(* Logix 5000 project; controller Savage_Saw vendor 1 type 14 code 152 rev 33.11; software revision 33.04 *)

TASK MainTask (continuous, watchdog 500 ms) : MainProgram

MODULES
   Local : vendor 1 type 14 code 152 (PointIO 0, rev 33.11)
      Kane : vendor 590 type 43 code 5 (Ethernet 192.168.1.11, rev 1.1, StandardDataDriven RPI 20 ms)
      Discrete_IO : Embedded (PointIO 1, rev 33.11, Output RPI 20 ms)
END_MODULES

TYPE Kane_OUT_DATA1 :
STRUCT
   Unassigned_Var_Table_12 : REAL;
   Unassigned_Var_Table_13 : REAL;
   Unassigned_Var_Table_14 : REAL;
   Unassigned_Var_Table_15 : REAL;
   Unassigned_Var_Table_16 : REAL;
   Unassigned_Var_Table_17 : REAL;
   Unassigned_Var_Table_18 : REAL;
   Unassigned_Var_Table_19 : REAL;
   Unassigned_Var_Table_20 : REAL;
   Unassigned_Var_Table_21 : REAL;
END_STRUCT
END_TYPE

TYPE RMC_IN :
STRUCT
   xCutStatus : DINT;
   yBedStatus : DINT;
   zDepthStatus : DINT;
   xCutPosition : REAL;
   yBedPosition : REAL;
   zDepthPosition : REAL;
END_STRUCT
END_TYPE

TYPE RMC_OUT :
STRUCT
   xCutPosnCommand : REAL;
   yBedPosnCommand : REAL;
   zDepthPosnCommand : REAL;
   xCutVelocity : REAL;
   yBedVelocity : REAL;
   zDepthVelocity : REAL;
END_STRUCT
END_TYPE

VAR_GLOBAL   (* controller tags *)
   RMC_Busy : BOOL;
   RMC_In : RMC_IN := (xCutStatus := 67154500, yBedStatus := 67117633, zDepthStatus := 67121732, xCutPosition := 15.000001, yBedPosition := 10.0, zDepthPosition := 18.928001);
   RMC_Out : RMC_OUT := (xCutPosnCommand := 9.999, yBedPosnCommand := 2.2, zDepthPosnCommand := 3.3, xCutVelocity := 4.4, yBedVelocity := 5.5, zDepthVelocity := 69.6);
   RMC_SendRequest : BOOL;
END_VAR

PROGRAM MainProgram   (* main routine RMC *)

ROUTINE RMC   (* ladder *)
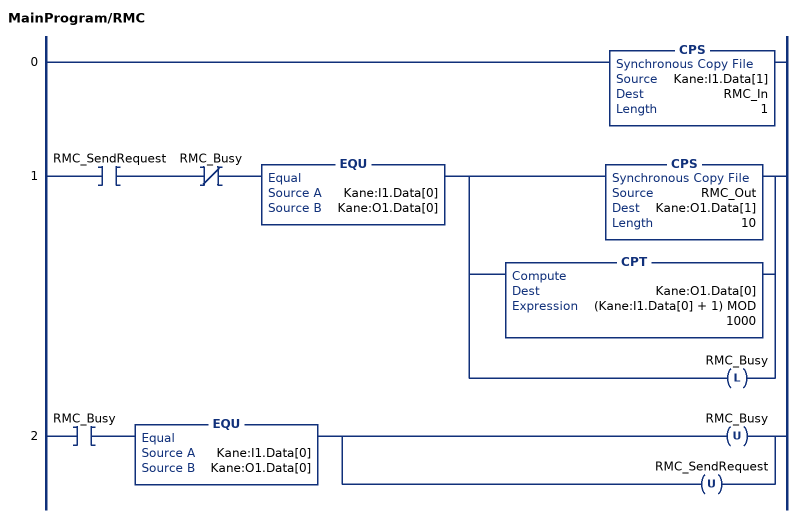
   0: CPS(Kane:I1.Data[1],RMC_In,1);
   1: XIC(RMC_SendRequest)XIO(RMC_Busy)EQU(Kane:I1.Data[0],Kane:O1.Data[0])[CPS(RMC_Out,Kane:O1.Data[1],10) ,CPT(Kane:O1.Data[0],(Kane:I1.Data[0] + 1) MOD 1000) ,OTL(RMC_Busy) ];
   2: XIC(RMC_Busy)EQU(Kane:I1.Data[0],Kane:O1.Data[0])[OTU(RMC_Busy) ,OTU(RMC_SendRequest) ];
END_ROUTINE
END_PROGRAM
